FUNCTION_BLOCK stateMachine
VAR_INPUT

	stBase             : REFERENCE TO stationBase;	// Базова структура на станция  
	activeEMG          : BOOL;                      // Има активен safety стоп
	
	depClear           : BOOL;
	syncClear          : BOOL;

	
	
END_VAR
VAR_OUTPUT
END_VAR


VAR
	stCurrentState     : DINT;  			        // Текущо състояние на станцията
	startUp            : BOOL := FALSE;    		    // Флаг който се сетва за 1 цикъл при първо извикване 
	statePass		   : BOOL; 						// Вече има избран следващ state
	depPass            : BOOL; 						// Depandancy е било изпълнено за даденият state
	depSyncPass		   : BOOL;                    // Всички завицещи от текущият state, други станций са били sync-нати
	stationStop		   : BOOL; 				        // Станцията е спряна
	depActive          : BOOL;                      // Станцията изчаква друга
	syncActive         : BOOL;                      // Станцията sync-ва друга
	syncArr            : ARRAY [0..Consts.MAX_SYNC_STATIONS] OF INT; 
	depCount           : INT;                       // Общ брой на dependency-ta към други станий в текущият state
	depIndex           : INT;                       // Индек за адресиране на dependency в syncArr
	stTimer		       : TON;						// Всяки state има по един таймер
	stErrTimer         : TON;                       // И по един за генериране на грешка 
	startTimer         : BOOL;                      // Битове за старт на таймерите
	startErrTimer      : BOOL;
	stTime             : TIME;                      // Време на stTimer-a - задава се от stаteDalay
	stErrTime          : TIME;                      // Време за stErrТimer-a - задава се от timeOutError
	io				   : ioControl;                 // Дефинира няколко метода за работа с IO
	tempState          : DINT;                      // Запазва некущото състояни за step mode
	stepModeActive     : BOOL; 						// Активен е стъпков режим
	debugTimer         : TON;
	debugTImerIN       : BOOL;

END_VAR


// Тази част на FB-то никога няма да се изпълни (и кода в нея)

METHOD PRIVATE cycle
VAR_INPUT
	
	ioImage            : ANY;                           // ioImage за станцията 
	
END_VAR

VAR 
	ioImageIndex    : POINTER TO DINT;                 // показва началото на IO Image структурата
	ioStruct		: POINTER TO imageIO;              // текуща структура - една IO точка (DI или DO)
	points 			: DINT;							   // брой на входове и изходи в дадената стация
END_VAR

// Служи за упр. на стъпковата машина (в случея Switch Case блок)
// Грижи се за правилното упр. на сигнали от Staion Base

// Станцията е на автоматичен режим и е активна
IF stBase.AutoMode AND stBase.ToggleEnable THEN
	
	stBase.Disabled := FALSE;
	
	// Индекса за dependency-та се нулара всеки цикъл (изпползва се в dependencySync)
	depIndex        := 0;
		
	// При първо извикване станцията преминава в стартово състояние
	IF NOT startUp THEN
		startUp 			 	   	 := TRUE;
		stBase.Busy 	      	 	 := FALSE;
		stBase.Ready		 	 	 := FALSE;
		stBase.Error    	  		 := FALSE;
		stBase.LastState      		 := Consts.ST_START_UP;
		stBase.CurrentState   		 := Consts.ST_START_UP;
		stBase.Error          		 := FALSE;
		stBase.LastErrorState        := Consts.ST_NULL;
		stBase.DoInit         		 := FALSE;
		stBase.DoStart        		 := FALSE;
		stBase.DoStop        		 := FALSE;
		stBase.DependencyState       := Consts.NO_DEPENDENCY;	
		stCurrentState 				 := Consts.ST_START_UP;
		tempState 				     := Consts.ST_NULL;
		depCount 				     := 0;
		depActive                    := FALSE;
		syncActive                   := FALSE;
		statePass 			   		 := FALSE;
		depPass 				     := FALSE;
		depSyncPass 			     := FALSE;
		MEMSET(ADR(syncArr), 0, SIZEOF(syncArr));

	END_IF
	
	// Без оглед на текущото състояние се задава състояние на стоп
    // Ако има започанала някаква манупулация тя ще завърши 

	IF stBase.DoStop THEN
	
		stBase.DoStop             := FALSE;
		stationStop               := TRUE; 
		stBase.Busy 	      	  := FALSE;
		stBase.Ready		 	  := FALSE;
		stBase.Error              := FALSE;
		stepModeActive            := FALSE;
		depCount 				  := 0;
		depActive                 := FALSE;
		syncActive                := FALSE;
		statePass 			      := FALSE;
		depPass 				  := FALSE;
		depSyncPass 			  := FALSE;		
		stBase.CurrentState       := Consts.ST_STOP;
		tempState 				  := Consts.ST_NULL;
	
	END_IF
	
	// Когато станцията е спряла или е имало грешка при командта RESTART от HMI (DoInt)
	// станцията се инициализира
	IF  stBase.DoInit THEN
		
	    stBase.DoInit                := FALSE;
		stBase.Error                 := FALSE;
		stationStop    			     := FALSE;
		statePass 			   		 := FALSE;
		stBase.DoConfirmDependency   := FALSE;
		depCount 				     := 0;
		depActive                    := FALSE;
		syncActive                   := FALSE;
		statePass 			   		 := FALSE;
		depPass 				     := FALSE;
		depSyncPass 			     := FALSE;		
		stBase.DependencyState       := Consts.NO_DEPENDENCY;	
		stBase.LastErrorState        := Consts.ST_NULL;
		stBase.CurrentState          := Consts.ST_INIT;
        MEMSET(ADR(syncArr), 0, SIZEOF(syncArr));
	ELSE
		stBase.DoInit                := FALSE;
	END_IF
	
	// Има активен safety предпазен стоп
	IF activeEMG THEN
			
		stBase.DoConfirmDependency   := FALSE;
		statePass 			   		 := FALSE;
		depPass 				     := FALSE;
		depSyncPass 			     := FALSE;		
		depCount 				     := 0;
		depActive                    := FALSE;
		syncActive                   := FALSE;
		stBase.DependencyState       := Consts.NO_DEPENDENCY;
		stepModeActive     		     := FALSE;
		tempState 				     := Consts.ST_NULL;
		startTimer       		     := FALSE;
		startErrTimer                := FALSE;
		stBase.CurrentState          := Consts.ST_EMG;
		stCurrentState               := Consts.ST_EMG;
		MEMSET(ADR(syncArr), 0, SIZEOF(syncArr));
	
	END_IF
	
	IF NOT stBase.Error AND NOT stationStop THEN
		IF stCurrentState = Consts.ST_READY OR stCurrentState = Consts.ST_STEP_BLOCK THEN	
			stBase.Ready := TRUE;
			stBase.Busy  := FALSE;	
		ELSE
			stBase.Ready := FALSE;
			stBase.Busy  := TRUE;			
		END_IF
	ELSE
		stBase.Ready := FALSE;
		stBase.Busy  := FALSE;
	END_IF
	
	// Правене на преход от към ново състояние
	IF stCurrentState <> stBase.CurrentState THEN
		
		startTimer       := FALSE;
		startErrTimer    := FALSE;
		statePass 		 := FALSE;
		depPass 		 := FALSE;
		depSyncPass 	 := FALSE;
		
		stBase.DependencyState       := Consts.NO_DEPENDENCY;
		
		IF stBase.NextStep or stepModeActive THEN
			IF  stBase.CurrentState <> Consts.ST_STEP_BLOCK THEN
				stepModeActive       := TRUE;                 // Активен е спъпков режим
				stBase.NextStep      := FALSE;
				tempState            := stBase.CurrentState;
				stBase.CurrentState  := Consts.ST_STEP_BLOCK;
				stCurrentState       := Consts.ST_STEP_BLOCK;
			END_IF
		ELSE
			stBase.LastState := stCurrentState;
			stCurrentState   := stBase.CurrentState;        // Следващ state при автоматичрн режим
		END_IF
		
	END_IF
	
	IF stCurrentState = Consts.ST_STEP_BLOCK AND stBase.NextStep THEN
		stBase.CurrentState  := tempState; 	
		stCurrentState       := tempState;
		stBase.NextStep      := FALSE;	
		statePass 			 := FALSE;
		depPass 			 := FALSE;
		depSyncPass 	     := FALSE;		
	END_IF
	
	// При активен съпков режим може да се продължи към автоматичен
	IF stepModeActive AND stBase.DoStart THEN
		 stBase.CurrentState  := tempState; 	
		 stCurrentState       := tempState;
		 stBase.DoStart       := FALSE;
		 stepModeActive       := FALSE;	
		 statePass 			  := FALSE;	
		 depPass 			  := FALSE;
		 depSyncPass 		  := FALSE;		 
	END_IF

	
	// Таймери за state-та - един за общо ползване и един за ген. на грешка
	stTimer   (IN := startTimer,    PT := stTime);
	stErrTimer(IN := startErrTimer, PT := stErrTime);
	

    // Когато станцията е спяла тогава може да се сетват и ресетват входове и изходи
	// Чрез ANY pointer и малко аритметика се адресира структура по структура и се проверява
	// дали трябва да се сетне дадено IO 
	IF stationStop THEN

		points         := ioImage.diSize / SIZEOF(imageIO);     // брой IO points за станция
		ioImageIndex   := ioImage.pValue;                       // стартов адрес на структурата
	
		WHILE points > 0 DO                                     // адрес на imageIO 
			
			ioStruct := ioImageIndex;  
                         
			IF ioStruct^.iType = ioType.INPUT_BIT THEN          // updata на pointa ако е вход
				ioStruct^.stIO := io.getX(ioStruct^);
		
			ELSIF ioStruct^.iType = ioType.OUTPUT_BIT THEN	
				IF ioStruct^.stIO THEN
					io.setY(ioStruct^);
				ELSE 
					io.rstY(ioStruct^);
				END_IF
			END_IF
		
			ioImageIndex := ioImageIndex + SIZEOF(imageIO);      // dec -  следващ IO point
			points       := points - 1;
		END_WHILE
	END_IF
			
ELSE
	// Станцията е изключена
	stBase.Disabled := TRUE;	
	startUp         := TRUE;
	
END_IF
END_METHOD

METHOD PROTECTED depNextState
VAR_INPUT
	
	station			: REFERENCE TO stationBase;       
	dep 			: DINT;  
    newState 		: DINT;                                             

END_VAR


// Ако има сигнализарано dependency от depSignal, веднага се прави преход
// към зададеният state. Всички останли dependency-та, (ако имa) се изчистват
// Тоест тази метод е с по-висок приоритет от depSync и depWait

IF  station.DependencyState = dep AND stCurrentState = stBase.CurrentState THEN
	
	MEMSET(ADR(syncArr), 0, SIZEOF(syncArr));
	syncActive       := FALSE;
	depActive        := FALSE;
	nextState(newState);

END_IF
END_METHOD

METHOD PROTECTED depSignal
VAR_INPUT
		
	dep 		: DINT;	

END_VAR

// Сетва dependency, но не блокира на него какво в depWait.
// Отново има място само за едно на state.
// Изчиства се автоматично при преминаване в следващият state

IF stBase.DependencyState = Consts.NO_DEPENDENCY AND stCurrentState = stBase.CurrentState THEN
	stBase.DependencyState      := dep;
END_IF
END_METHOD

METHOD PROTECTED depSync
VAR_INPUT
	
	station			: REFERENCE TO stationBase;       // станция от която е извикан dependencyWait
	dep 			: DINT;                           // какво dependency е сетнато

// Трябва dependency-то което се очаква и това което sync-ва да са еднакви!
// Иначе ще има dead-lock в текущите състояние и на двете станций.                         


END_VAR

// Метода потвърждата дадето dependency от друга станция.
// В един state може да има до 64 Sync извиквания - докато всичките
// такива не се изпълнят станцията няма да мине в следващ state.

IF stCurrentState = stBase.CurrentState AND NOT depSyncPass THEN
	syncActive    := TRUE;                        // спира се възможноста за преход в друг state
	
	// Когато за първи път извика метода даденото dependency се макрира като вече отчетено
	// Брояча на dependency-та се увеличава. Така се знае колко трябва да се изпълнят за дадения state
	// и чак след като всички се sync-ват и може да се премине в следващ state
	IF syncArr[depIndex] = 0 THEN
	
		syncArr[depIndex] := Consts.DEP_PASS;
		depCount          := depCount + 1;

	// Има маркирано dependency и на него се чака в друга станция
	// Другата станция се "освобождава" а тук брояча на dependency-та се намалява - има sync-нато dependency
	ELSIF (syncArr[depIndex] = Consts.DEP_PASS AND station.DependencyState = dep) OR syncClear THEN
	
		syncArr[depIndex]       := Consts.SYNC_CONFIRM;
		station.DependencyState := Consts.NO_DEPENDENCY;
		depCount 		        := depCount - 1;
	
	END_IF
	
		depIndex          := depIndex + 1;
	
END_IF
END_METHOD

METHOD PROTECTED depWait

VAR_INPUT
	
     dep			: DINT;          // dependency което трябва да се Sync-не от друга станция

END_VAR

// Сетва определено dependency в stationBase
// Станцията не може да премине в друг state докато това dependency 
// не се потвърди от depenencySync ф-я.
// В един state може да има само едно извикване на dependencyWait, защото
// в stationBase има място само за едно.


IF stBase.DependencyState = Consts.NO_DEPENDENCY AND NOT depActive AND stCurrentState = stBase.CurrentState AND NOT depPass THEN
	stBase.DependencyState      := dep;
	depActive                   := TRUE;
ELSIF (stBase.DependencyState = Consts.NO_DEPENDENCY AND depActive) OR depClear THEN
	depActive 					:= FALSE;
	depClear                    := FALSE;
	depPass                     := TRUE;
END_IF
END_METHOD

METHOD PROTECTED nextState
VAR_INPUT
	
	nextState 		:DINT;                     // Следващо състояние

END_VAR

debugTimer(IN := debugTimerIN, PT := T#2S);

// Ако няма грешка или активно dependency или ако няма sync-ване

IF NOT stBase.Error AND NOT stationStop AND NOT depActive AND NOT syncActive AND NOT activeEMG AND NOT statePass THEN 

	IF DEBUG.noErrors THEN
		debugTimerIN := TRUE;
		IF debugTimer.Q THEN
		    stBase.CurrentState    := nextState;
			statePass 			   := TRUE;	
			debugTimerIN           := FALSE;
		END_IF	
	ELSE
  	    stBase.CurrentState    := nextState;
	    statePass 			   := TRUE;
	END_IF
	
END_IF
	

// При активно dependency, може да се премине в следващ state
// само ако брояча на dependency-та за дадения state e нула
// Това значи че те всички са sync-нати

IF syncActive AND depCount = 0  AND NOT depActive THEN

// Изчиства се масива в който е бил "маркиран" статута на 
// dependency-та в stata-та	

    MEMSET(ADR(syncArr), 0, SIZEOF(syncArr));
	
	syncActive             := FALSE;
    stBase.CurrentState    := nextState;
	statePass 			   := TRUE;
	depSyncPass            := TRUE;
		
END_IF
END_METHOD

METHOD PROTECTED setDisplayState
VAR_INPUT
	
	displayState		: DINT;         // състояние за виз. на HMI

END_VAR

// Просто актуализира променлива за displayState

IF displayState <> Consts.ST_NULL THEN
	stBase.DisplayState    := displayState;
END_IF
END_METHOD

METHOD PROTECTED setError
VAR_INPUT
		
	errState    :   DINT;       // състоянието за дадената грешка

END_VAR

// Този метод всъщност просто преминава към зададеното му състояние
// Разликата от nextState е че сетва и бит Error в stationBase
// Прехода се прави веднаги без да се отчита dependency 
IF NOT stBase.Error AND NOT stationStop AND stCurrentState = stBase.CurrentState AND NOT DEBUG.noErrors THEN 
	stBase.CurrentState    := errState;
	stBase.LastErrorState  := errState;
	stBase.Error           := TRUE;
    Global.machError       := TRUE;    

END_IF
END_METHOD

METHOD PROTECTED setStateVars
VAR_INPUT
	
    img            : ANY;       // ioImage за станцията 	

END_VAR
VAR_IN_OUT
	sv			: DINT; 		 // state var - текущо състояние
END_VAR

// Текущото състояние на станцията се записва като променлива 
// в stateMachine, за да могат всички методи да имат достъп до нея
// Изпълнява се упр. цикъл, update-ва се stateVar и се изпълнява главния switch case
// на станцията.

THIS^.stCurrentState := sv;

cycle(img);

sv := This^.stCurrentState;
END_METHOD

METHOD PROTECTED stateDelay : BOOL
VAR_INPUT

	t       : TIME;         // време на stTimer-a	

END_VAR

// Когато се извика тази ф-я стартира таймер
// Той е един за всяки state и е ощо ползване
// Min. времето е поне 10ms
// Ресетва се при преминаване в следващ state

IF t > T#10MS AND NOT startTimer THEN
	stTime     := t;
	startTimer := TRUE;	
END_IF


IF stTimer.Q THEN
	stateDelay   := TRUE;
ELSE
	stateDelay   := FALSE;
END_IF
END_METHOD

METHOD PROTECTED timeOutError
VAR_INPUT
	
	t				: TIME;      // време след което се ген. преминава в грешка
	stErr           : DINT;      // сътояние на грешката 

END_VAR
// Когато се извика тази ф-я стартира таймер
// След изтичането му се преминава в състояние не грешка
// Min. времето е поне 10ms
// Ресетва се при преминаване в следващ state

IF t > T#10MS AND NOT startErrTimer AND NOT DEBUG.noErrors THEN
	stErrTime       := t;
	startErrTimer   := TRUE;	
END_IF


IF stErrTimer.Q THEN
	setError(stErr);
END_IF
END_METHOD

END_FUNCTION_BLOCK

(* stored: Version 1.1.0.1, ProductVersion 3.1.4024.3
   POU stateMachine: Id {cf3e709c-ead8-4319-8a8c-bafc90188536}, SpecialFunc None
   Method cycle: Id {05fb74c1-c6fb-48aa-97e1-fcb7c37d362f}
   Method depNextState: Id {7cd1e24c-6af1-42e7-84f0-771d8a513191}
   Method depSignal: Id {2573fba1-3e06-4376-bb55-5f33c87a4f12}
   Method depSync: Id {f01e89e7-9750-4444-9e99-be7ba4e68ec9}
   Method depWait: Id {c80b042d-6ec4-4378-ab99-f053f7ac1503}
   Method nextState: Id {b075e5c8-0934-491b-949f-0a60771edadc}
   Method setDisplayState: Id {1e5fce71-9784-4cc8-8d2f-af555a57ce71}
   Method setError: Id {ad1afc0c-b58e-47c1-bd8e-0ba96e2df6a6}
   Method setStateVars: Id {63224c19-553c-4b8c-8137-1d45bca60bd0}
   Method stateDelay: Id {240fde62-c5f9-4152-9a0d-553b967184eb}
   Method timeOutError: Id {686753c6-058e-408e-84a2-c5394200967e} *)
